(* CODESYS project AgitatorSequence.xml

Project tree, tasks and I/O mapping:
  function block AgitatorSequence [SFC]
*)

// AgitatorSequence
FUNCTION_BLOCK AgitatorSequence
// This Sequential Function Chart function block is for sequencing one agitator cycle each time it is triggered.
VAR_INPUT
	Trigger: 			BOOL; 				// Trigger bit to start the agitator sequence.
	ReverseTime: 		TIME; 				// Agitator cycle time spent in reverse motion.
	DwellTime: 			TIME;   			// Agitator cycle time spent dwelling between reverse-forward motion.
	ForwardTime: 		TIME; 				// Agitator cycle time spent in forward motion.
END_VAR
VAR_OUTPUT
	Complete: 			BOOL; 				// Output bit that pulses when the sequence completes.
	Forward: 			BOOL; 				// Output for motor forward command.
	Reverse: 			BOOL; 				// Output for motor reverse command.
	Dwell: 				BOOL; 				// Output for when dwelling between directions.
	Agitating: 			BOOL; 				// Output bit that is on while the agitating sequence is active.
END_VAR
VAR
END_VAR

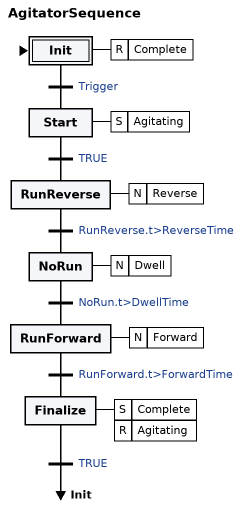
INITIAL_STEP Init:
    Complete(R);
END_STEP
TRANSITION FROM Init TO Start
    := Trigger;
END_TRANSITION
STEP Start:
    Agitating(S);
END_STEP
TRANSITION FROM Start TO RunReverse
    := TRUE;
END_TRANSITION
STEP RunReverse:
    Reverse(N);
END_STEP
TRANSITION FROM RunReverse TO NoRun
    := RunReverse.t>ReverseTime;
END_TRANSITION
STEP NoRun:
    Dwell(N);
END_STEP
TRANSITION FROM NoRun TO RunForward
    := NoRun.t>DwellTime;
END_TRANSITION
STEP RunForward:
    Forward(N);
END_STEP
TRANSITION FROM RunForward TO Finalize
    := RunForward.t>ForwardTime;
END_TRANSITION
STEP Finalize:
    Complete(S);
    Agitating(R);
END_STEP
TRANSITION FROM Finalize TO Init
    := TRUE;
END_TRANSITION

END_FUNCTION_BLOCK
